// Monitors the baseplate chiller from the flow sensor
FUNCTION_BLOCK FB_BaseplateChiller
VAR_INPUT
    bAmphosOn : BOOL; // Whether the amphos is turned on
	bBaseplateChillerFlow : BOOL; // Signal from the flow sensor. Normally high.
	bMasterLatchReset : BOOL; //Master latched error reset
END_VAR
VAR_OUTPUT
	{attribute 'pytmc' := '
		pv: ERROR
		io: i
		field: OSV MAJOR
		field: ZSV NO_ALARM
		field: ZNAM OK
		field: ONAM ERROR
	'}
	bError : BOOL; // Whether an error was detected. Should latch until reset
END_VAR
VAR
END_VAR

(* Latch error if the baseplate chiller flow detects an error *)
IF bAmphosOn AND NOT bBaseplateChillerFlow THEN
	bError := TRUE;
END_IF

IF bMasterLatchReset THEN
	bError := FALSE;
END_IF

// Reset latched errors
METHOD Reset
VAR_INPUT
END_VAR
bError := FALSE;
END_METHOD

END_FUNCTION_BLOCK

(* stored: Version 1.1.0.1, ProductVersion 3.1.4024.6
   POU FB_BaseplateChiller: Id {f1c4e0fa-ca2a-4b3d-bba0-0ee01f0d5f92}, SpecialFunc None
   Method Reset: Id {40d91e9c-2d15-4c66-8abe-ad4cf84eb069} *)
